// TIA Portal V17 export
// export: Created 2024-08-09T12:53:17.0936989Z, ExportSetting WithDefaults, DisplayName Totally Integrated Automation Portal, DisplayVersion V17 Update 7, DisplayName TIA Portal Openness, DisplayVersion V17 Update 7, DisplayName TIA Portal Version Control Interface, DisplayVersion V17, DisplayName STEP 7 Professional, DisplayVersion V17 Update 7, DisplayName STEP 7 Safety, DisplayVersion V17 Update 6, DisplayName WinCC Professional, DisplayVersion V17 Update 7
TYPE "S_Zone_Suiv_Lot"
// stored: IsFailsafeCompliant false
   STRUCT
      Occupee { ExternalAccessible := 'False'; ExternalVisible := 'False'; ExternalWritable := 'False'} : Bool;   // Flag indiquant zone de suivi occupee
      Taches { ExternalAccessible := 'False'; ExternalVisible := 'False'; ExternalWritable := 'False'} : Array[0.."Nbr_Max_Tache"] of "S_Tache";   // Liste des taches
   END_STRUCT;
END_TYPE
